{attribute 'linkalways'}
{attribute 'hide_all_locals'}
FUNCTION_BLOCK ValueLtime EXTENDS ValueLtimeRead IMPLEMENTS Value
VAR
END_VAR

METHOD SetFromType : BOOL
VAR_INPUT
	source : __SYSTEM.AnyType;
END_VAR
SetFromType := ConvertAnyType(source, thisAnyType);
END_METHOD

METHOD SetFromString : BOOL
VAR_INPUT
	value : T_MaxString;
END_VAR
thisValue := STRING_TO_LTIME(value);

SetFromString := TRUE;
END_METHOD

METHOD Set : BOOL
VAR_INPUT
	source : ANY;
END_VAR
Set := ConvertAnyType(source, thisAnyType);
END_METHOD

END_FUNCTION_BLOCK

(* stored: Version 1.1.0.1
   POU ValueLtime: Id {59dd599f-aa8a-43d0-b0ea-890c87db26aa}, SpecialFunc None
   Method SetFromType: Id {67daa6c9-022e-4330-9f7b-23dadc3700a6}
   Method SetFromString: Id {c0dee8ad-474f-46d4-b03d-f1879a21b722}
   Method Set: Id {0118e07c-9964-41e2-9326-ccacde6cf146} *)
